PROGRAM MAIN
VAR
END_VAR

END_PROGRAM

(* stored: Version 1.1.0.1, ProductVersion 3.1.4024.9
   POU MAIN: Id {1b2d04b9-4854-48f3-a572-b958903ec784}, SpecialFunc None *)
